(* IEC 61131-3 sources: brOscatLib/oscatBasic_tests/main, 2 files *)

(* ---- LocalVariables.var ---- *)
VAR
    testReporter : utTestReporter; (*Calculator for summaries of tests*)
END_VAR

(* ---- main.st ---- *)
PROGRAM _CYCLIC
    (**)
    testReporter(Results:=ADR(gResults), Size := SIZEOF(gResults) / SIZEOF(gResults[0]));
END_PROGRAM
